PROGRAM EXAMPLE //Example program for a specific application 
VAR

END_VAR

//Program any specific code or safety code for an specific application

END_PROGRAM

(* stored: Version 1.1.0.1, ProductVersion 3.1.4024.5
   POU EXAMPLE: Id {4bdeebc0-15d8-4790-97d0-e9c4239d121c}, SpecialFunc None *)
